// TIA Portal V17 export
// export: Created 2022-03-12T16:05:28.2107683Z, ExportSetting WithDefaults, DisplayName Totally Integrated Automation Portal, DisplayVersion V17, DisplayName TIA Portal Openness, DisplayVersion V17, DisplayName TIA Portal Version Control Interface, DisplayVersion V17, DisplayName STEP 7 Professional, DisplayVersion V17, DisplayName STEP 7 Safety, DisplayVersion V17, DisplayName WinCC Advanced / Unified PC, DisplayVersion V17
FUNCTION_BLOCK "EM01_01_EventControl"   // FB31661, LAD
TITLE = EM01_01_EventControl
{ S7_Optimized_Access := 'TRUE' }
AUTHOR : tech.team.motioncontrol@siemens.com
FAMILY : CPG
VERSION : 1.1
// Support: tech.team.motioncontrol@siemens.com
// stored: AutoNumber true, IsIECCheckEnabled false, IsRetainMemResEnabled false, MemoryReserve 100, SetENOAutomatically false, UDAEnableTagReadback false
   VAR
      instEventMgr_Alarm { ExternalAccessible := 'False'; ExternalVisible := 'False'; ExternalWritable := 'False'; S7_SetPoint := 'True'} : "CPG_EventManager";   // instance FB - Event Manager - Alarm Events
      instEventMgr_Warning { ExternalAccessible := 'False'; ExternalVisible := 'False'; ExternalWritable := 'False'; S7_SetPoint := 'True'} : "CPG_EventManager";   // instance FB - Event Manager - Warning Events
      instEventMgr_Status { ExternalAccessible := 'False'; ExternalVisible := 'False'; ExternalWritable := 'False'; S7_SetPoint := 'True'} : "CPG_EventManager";   // instance FB - Event Manager - Status Events
      instStatus_AlarmNotReset { ExternalAccessible := 'False'; ExternalVisible := 'False'; ExternalWritable := 'False'; S7_SetPoint := 'True'} : "CPG_Event";   // instance FB - PackML Event - Alarms not reset
      statEventMgr_Cmd_Reset { ExternalAccessible := 'False'; ExternalVisible := 'False'; ExternalWritable := 'False'} : Bool;   // Reset Cmd for all event managers
      statEventMgr_Cmd_Clear1stFlt { ExternalAccessible := 'False'; ExternalVisible := 'False'; ExternalWritable := 'False'} : Bool;   // Clear 1st Fault Cmd for all event managers
      statEventMgr_Clear1stFlt_OS { ExternalAccessible := 'False'; ExternalVisible := 'False'; ExternalWritable := 'False'} : Bool;   // Clear 1st Fault Cmd - One shot
   END_VAR
   VAR_TEMP   // added for the SCL form of the ladder/FBD networks
      _w1 : Bool;
      _w2 : Bool;
   END_VAR
BEGIN

REGION Network 1: ** STATE MODEL REPORTING STATUS ****
END_REGION

REGION Network 2: *** Call the PackML Module Initialize Logic ***
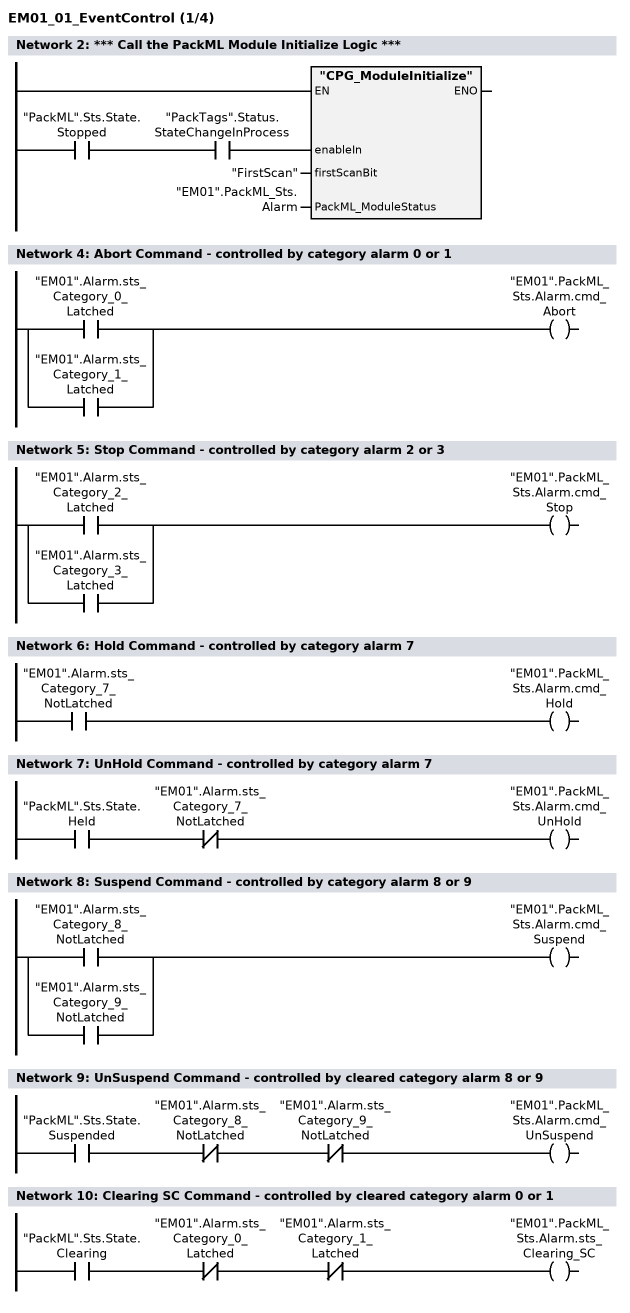
   RUNG wire#powerrail
      "CPG_ModuleInitialize"(enableIn := wire#w1, firstScanBit := "FirstScan", PackML_ModuleStatus := "EM01".PackML_Sts.Alarm)
   END_RUNG
   RUNG wire#powerrail
      Contact( "PackML".Sts.State.Stopped )
      Contact( "PackTags".Status.StateChangeInProcess )
   END_RUNG wire#w1
   // the same network as SCL:
   "CPG_ModuleInitialize"(enableIn := "PackML".Sts.State.Stopped AND "PackTags".Status.StateChangeInProcess,
                          firstScanBit := "FirstScan",
                          PackML_ModuleStatus := "EM01".PackML_Sts.Alarm);
END_REGION

REGION Network 3: Begin the LOGIC section.
END_REGION

REGION Network 4: Abort Command - controlled by category alarm 0 or 1
   RUNG wire#powerrail
      Contact( "EM01".Alarm.sts_Category_0_Latched )
      wire#w1
      Coil( "EM01".PackML_Sts.Alarm.cmd_Abort )
   END_RUNG
   RUNG wire#powerrail
      Contact( "EM01".Alarm.sts_Category_1_Latched )
   END_RUNG wire#w1
   // the same network as SCL:
   "EM01".PackML_Sts.Alarm.cmd_Abort := "EM01".Alarm.sts_Category_0_Latched OR "EM01".Alarm.sts_Category_1_Latched;
END_REGION

REGION Network 5: Stop Command - controlled by category alarm 2 or 3
   RUNG wire#powerrail
      Contact( "EM01".Alarm.sts_Category_2_Latched )
      wire#w1
      Coil( "EM01".PackML_Sts.Alarm.cmd_Stop )
   END_RUNG
   RUNG wire#powerrail
      Contact( "EM01".Alarm.sts_Category_3_Latched )
   END_RUNG wire#w1
   // the same network as SCL:
   "EM01".PackML_Sts.Alarm.cmd_Stop := "EM01".Alarm.sts_Category_2_Latched OR "EM01".Alarm.sts_Category_3_Latched;
END_REGION

REGION Network 6: Hold Command - controlled by category alarm 7
   RUNG wire#powerrail
      Contact( "EM01".Alarm.sts_Category_7_NotLatched )
      Coil( "EM01".PackML_Sts.Alarm.cmd_Hold )
   END_RUNG
   // the same network as SCL:
   "EM01".PackML_Sts.Alarm.cmd_Hold := "EM01".Alarm.sts_Category_7_NotLatched;
END_REGION

REGION Network 7: UnHold Command - controlled by category alarm 7
   RUNG wire#powerrail
      Contact( "PackML".Sts.State.Held )
      I_Contact( "EM01".Alarm.sts_Category_7_NotLatched )
      Coil( "EM01".PackML_Sts.Alarm.cmd_UnHold )
   END_RUNG
   // the same network as SCL:
   "EM01".PackML_Sts.Alarm.cmd_UnHold := "PackML".Sts.State.Held AND NOT "EM01".Alarm.sts_Category_7_NotLatched;
END_REGION

REGION Network 8: Suspend Command - controlled by category alarm 8 or 9
   RUNG wire#powerrail
      Contact( "EM01".Alarm.sts_Category_8_NotLatched )
      wire#w1
      Coil( "EM01".PackML_Sts.Alarm.cmd_Suspend )
   END_RUNG
   RUNG wire#powerrail
      Contact( "EM01".Alarm.sts_Category_9_NotLatched )
   END_RUNG wire#w1
   // the same network as SCL:
   "EM01".PackML_Sts.Alarm.cmd_Suspend := "EM01".Alarm.sts_Category_8_NotLatched OR "EM01".Alarm.sts_Category_9_NotLatched;
END_REGION

REGION Network 9: UnSuspend Command - controlled by cleared category alarm 8 or 9
   RUNG wire#powerrail
      Contact( "PackML".Sts.State.Suspended )
      I_Contact( "EM01".Alarm.sts_Category_8_NotLatched )
      I_Contact( "EM01".Alarm.sts_Category_9_NotLatched )
      Coil( "EM01".PackML_Sts.Alarm.cmd_UnSuspend )
   END_RUNG
   // the same network as SCL:
   "EM01".PackML_Sts.Alarm.cmd_UnSuspend := "PackML".Sts.State.Suspended AND NOT "EM01".Alarm.sts_Category_8_NotLatched AND NOT "EM01".Alarm.sts_Category_9_NotLatched;
END_REGION

REGION Network 10: Clearing SC Command - controlled by cleared category alarm 0 or 1
   RUNG wire#powerrail
      Contact( "PackML".Sts.State.Clearing )
      I_Contact( "EM01".Alarm.sts_Category_0_Latched )
      I_Contact( "EM01".Alarm.sts_Category_1_Latched )
      Coil( "EM01".PackML_Sts.Alarm.sts_Clearing_SC )
   END_RUNG
   // the same network as SCL:
   "EM01".PackML_Sts.Alarm.sts_Clearing_SC := "PackML".Sts.State.Clearing AND NOT "EM01".Alarm.sts_Category_0_Latched AND NOT "EM01".Alarm.sts_Category_1_Latched;
END_REGION

REGION Network 11: Resetting SC Command - controlled by cleared category alarm 0-3
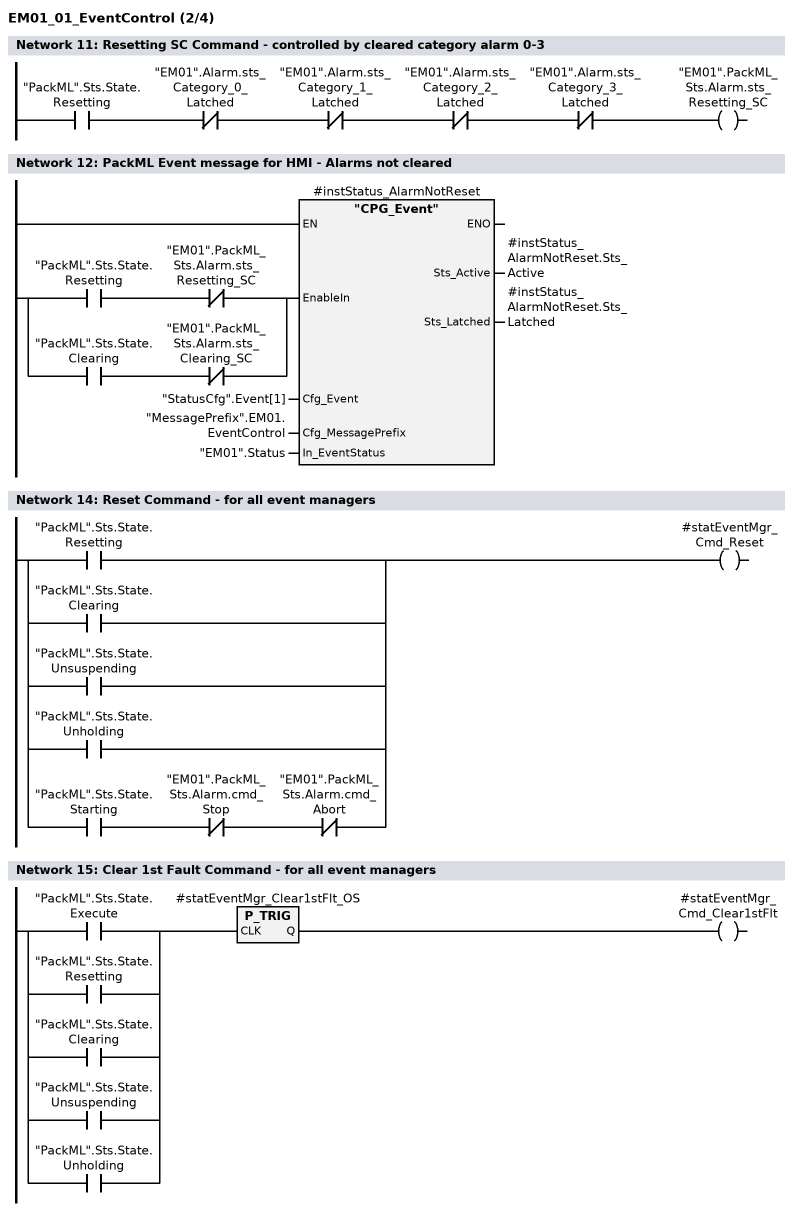
   RUNG wire#powerrail
      Contact( "PackML".Sts.State.Resetting )
      I_Contact( "EM01".Alarm.sts_Category_0_Latched )
      I_Contact( "EM01".Alarm.sts_Category_1_Latched )
      I_Contact( "EM01".Alarm.sts_Category_2_Latched )
      I_Contact( "EM01".Alarm.sts_Category_3_Latched )
      Coil( "EM01".PackML_Sts.Alarm.sts_Resetting_SC )
   END_RUNG
   // the same network as SCL:
   "EM01".PackML_Sts.Alarm.sts_Resetting_SC := "PackML".Sts.State.Resetting AND NOT "EM01".Alarm.sts_Category_0_Latched AND NOT "EM01".Alarm.sts_Category_1_Latched AND NOT "EM01".Alarm.sts_Category_2_Latched AND NOT "EM01".Alarm.sts_Category_3_Latched;
END_REGION

REGION Network 12: PackML Event message for HMI - Alarms not cleared
   RUNG wire#powerrail
      #instStatus_AlarmNotReset(EnableIn := wire#w1, Cfg_Event := "StatusCfg".Event[1], Cfg_MessagePrefix := "MessagePrefix".EM01.EventControl, In_EventStatus := "EM01".Status, Sts_Active => #instStatus_AlarmNotReset.Sts_Active, Sts_Latched => #instStatus_AlarmNotReset.Sts_Latched)
   END_RUNG
   RUNG wire#powerrail
      Contact( "PackML".Sts.State.Resetting )
      I_Contact( "EM01".PackML_Sts.Alarm.sts_Resetting_SC )
   END_RUNG wire#w1
   RUNG wire#powerrail
      Contact( "PackML".Sts.State.Clearing )
      I_Contact( "EM01".PackML_Sts.Alarm.sts_Clearing_SC )
   END_RUNG wire#w1
   // the same network as SCL:
   #instStatus_AlarmNotReset(EnableIn := ("PackML".Sts.State.Resetting AND NOT "EM01".PackML_Sts.Alarm.sts_Resetting_SC) OR ("PackML".Sts.State.Clearing AND NOT "EM01".PackML_Sts.Alarm.sts_Clearing_SC),   // "CPG_Event"
                           Cfg_Event := "StatusCfg".Event[1],
                           Cfg_MessagePrefix := "MessagePrefix".EM01.EventControl,
                           In_EventStatus := "EM01".Status,
                           Sts_Active => #instStatus_AlarmNotReset.Sts_Active,
                           Sts_Latched => #instStatus_AlarmNotReset.Sts_Latched);
END_REGION

REGION Network 13: *** EVENT CONTROL MANAGERS ***
END_REGION

REGION Network 14: Reset Command - for all event managers
   RUNG wire#powerrail
      Contact( "PackML".Sts.State.Resetting )
      wire#w1
      Coil( #statEventMgr_Cmd_Reset )
   END_RUNG
   RUNG wire#powerrail
      Contact( "PackML".Sts.State.Clearing )
   END_RUNG wire#w1
   RUNG wire#powerrail
      Contact( "PackML".Sts.State.Unsuspending )
   END_RUNG wire#w1
   RUNG wire#powerrail
      Contact( "PackML".Sts.State.Unholding )
   END_RUNG wire#w1
   RUNG wire#powerrail
      Contact( "PackML".Sts.State.Starting )
      I_Contact( "EM01".PackML_Sts.Alarm.cmd_Stop )
      I_Contact( "EM01".PackML_Sts.Alarm.cmd_Abort )
   END_RUNG wire#w1
   // the same network as SCL:
   #statEventMgr_Cmd_Reset := "PackML".Sts.State.Resetting OR "PackML".Sts.State.Clearing OR "PackML".Sts.State.Unsuspending OR "PackML".Sts.State.Unholding OR ("PackML".Sts.State.Starting AND NOT "EM01".PackML_Sts.Alarm.cmd_Stop AND NOT "EM01".PackML_Sts.Alarm.cmd_Abort);
END_REGION

REGION Network 15: Clear 1st Fault Command - for all event managers
   RUNG wire#powerrail
      Contact( "PackML".Sts.State.Execute )
      wire#w1
      P_Trig( #statEventMgr_Clear1stFlt_OS )
      Coil( #statEventMgr_Cmd_Clear1stFlt )
   END_RUNG
   RUNG wire#powerrail
      Contact( "PackML".Sts.State.Resetting )
   END_RUNG wire#w1
   RUNG wire#powerrail
      Contact( "PackML".Sts.State.Clearing )
   END_RUNG wire#w1
   RUNG wire#powerrail
      Contact( "PackML".Sts.State.Unsuspending )
   END_RUNG wire#w1
   RUNG wire#powerrail
      Contact( "PackML".Sts.State.Unholding )
   END_RUNG wire#w1
   // the same network as SCL:
   #_w1 := "PackML".Sts.State.Execute OR "PackML".Sts.State.Resetting OR "PackML".Sts.State.Clearing OR "PackML".Sts.State.Unsuspending OR "PackML".Sts.State.Unholding;
   #_w2 := #_w1 AND NOT #statEventMgr_Clear1stFlt_OS;   // rising edge
   #statEventMgr_Clear1stFlt_OS := #_w1;
   #statEventMgr_Cmd_Clear1stFlt := #_w2;
END_REGION

REGION Network 16: Call the Event Manager logic for EM alarms
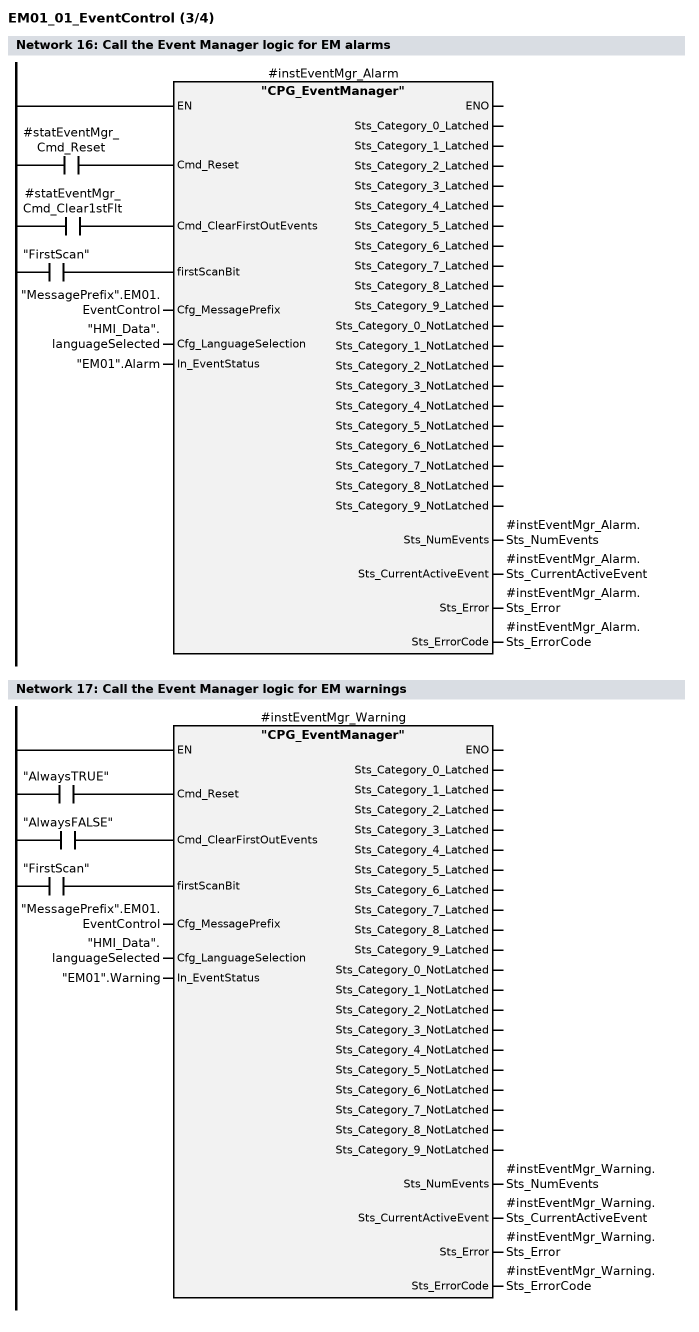
   RUNG wire#powerrail
      #instEventMgr_Alarm(Cmd_Reset := wire#w1, Cmd_ClearFirstOutEvents := wire#w2, firstScanBit := wire#w3, Cfg_MessagePrefix := "MessagePrefix".EM01.EventControl, Cfg_LanguageSelection := "HMI_Data".languageSelected, In_EventStatus := "EM01".Alarm, Sts_Category_0_Latched =>, Sts_Category_1_Latched =>, Sts_Category_2_Latched =>, Sts_Category_3_Latched =>, Sts_Category_4_Latched =>, Sts_Category_5_Latched =>, Sts_Category_6_Latched =>, Sts_Category_7_Latched =>, Sts_Category_8_Latched =>, Sts_Category_9_Latched =>, Sts_Category_0_NotLatched =>, Sts_Category_1_NotLatched =>, Sts_Category_2_NotLatched =>, Sts_Category_3_NotLatched =>, Sts_Category_4_NotLatched =>, Sts_Category_5_NotLatched =>, Sts_Category_6_NotLatched =>, Sts_Category_7_NotLatched =>, Sts_Category_8_NotLatched =>, Sts_Category_9_NotLatched =>, Sts_NumEvents => #instEventMgr_Alarm.Sts_NumEvents, Sts_CurrentActiveEvent => #instEventMgr_Alarm.Sts_CurrentActiveEvent, Sts_Error => #instEventMgr_Alarm.Sts_Error, Sts_ErrorCode => #instEventMgr_Alarm.Sts_ErrorCode)
   END_RUNG
   RUNG wire#powerrail
      Contact( #statEventMgr_Cmd_Reset )
   END_RUNG wire#w1
   RUNG wire#powerrail
      Contact( #statEventMgr_Cmd_Clear1stFlt )
   END_RUNG wire#w2
   RUNG wire#powerrail
      Contact( "FirstScan" )
   END_RUNG wire#w3
   // the same network as SCL:
   #instEventMgr_Alarm(Cmd_Reset := #statEventMgr_Cmd_Reset,   // "CPG_EventManager"
                       Cmd_ClearFirstOutEvents := #statEventMgr_Cmd_Clear1stFlt,
                       firstScanBit := "FirstScan",
                       Cfg_MessagePrefix := "MessagePrefix".EM01.EventControl,
                       Cfg_LanguageSelection := "HMI_Data".languageSelected,
                       In_EventStatus := "EM01".Alarm,
                       Sts_NumEvents => #instEventMgr_Alarm.Sts_NumEvents,
                       Sts_CurrentActiveEvent => #instEventMgr_Alarm.Sts_CurrentActiveEvent,
                       Sts_Error => #instEventMgr_Alarm.Sts_Error,
                       Sts_ErrorCode => #instEventMgr_Alarm.Sts_ErrorCode);
END_REGION

REGION Network 17: Call the Event Manager logic for EM warnings
   RUNG wire#powerrail
      #instEventMgr_Warning(Cmd_Reset := wire#w1, Cmd_ClearFirstOutEvents := wire#w2, firstScanBit := wire#w3, Cfg_MessagePrefix := "MessagePrefix".EM01.EventControl, Cfg_LanguageSelection := "HMI_Data".languageSelected, In_EventStatus := "EM01".Warning, Sts_Category_0_Latched =>, Sts_Category_1_Latched =>, Sts_Category_2_Latched =>, Sts_Category_3_Latched =>, Sts_Category_4_Latched =>, Sts_Category_5_Latched =>, Sts_Category_6_Latched =>, Sts_Category_7_Latched =>, Sts_Category_8_Latched =>, Sts_Category_9_Latched =>, Sts_Category_0_NotLatched =>, Sts_Category_1_NotLatched =>, Sts_Category_2_NotLatched =>, Sts_Category_3_NotLatched =>, Sts_Category_4_NotLatched =>, Sts_Category_5_NotLatched =>, Sts_Category_6_NotLatched =>, Sts_Category_7_NotLatched =>, Sts_Category_8_NotLatched =>, Sts_Category_9_NotLatched =>, Sts_NumEvents => #instEventMgr_Warning.Sts_NumEvents, Sts_CurrentActiveEvent => #instEventMgr_Warning.Sts_CurrentActiveEvent, Sts_Error => #instEventMgr_Warning.Sts_Error, Sts_ErrorCode => #instEventMgr_Warning.Sts_ErrorCode)
   END_RUNG
   RUNG wire#powerrail
      Contact( "AlwaysTRUE" )
   END_RUNG wire#w1
   RUNG wire#powerrail
      Contact( "AlwaysFALSE" )
   END_RUNG wire#w2
   RUNG wire#powerrail
      Contact( "FirstScan" )
   END_RUNG wire#w3
   // the same network as SCL:
   #instEventMgr_Warning(Cmd_Reset := "AlwaysTRUE",   // "CPG_EventManager"
                         Cmd_ClearFirstOutEvents := "AlwaysFALSE",
                         firstScanBit := "FirstScan",
                         Cfg_MessagePrefix := "MessagePrefix".EM01.EventControl,
                         Cfg_LanguageSelection := "HMI_Data".languageSelected,
                         In_EventStatus := "EM01".Warning,
                         Sts_NumEvents => #instEventMgr_Warning.Sts_NumEvents,
                         Sts_CurrentActiveEvent => #instEventMgr_Warning.Sts_CurrentActiveEvent,
                         Sts_Error => #instEventMgr_Warning.Sts_Error,
                         Sts_ErrorCode => #instEventMgr_Warning.Sts_ErrorCode);
END_REGION

REGION Network 18: Call the Event Manager logic for EM status
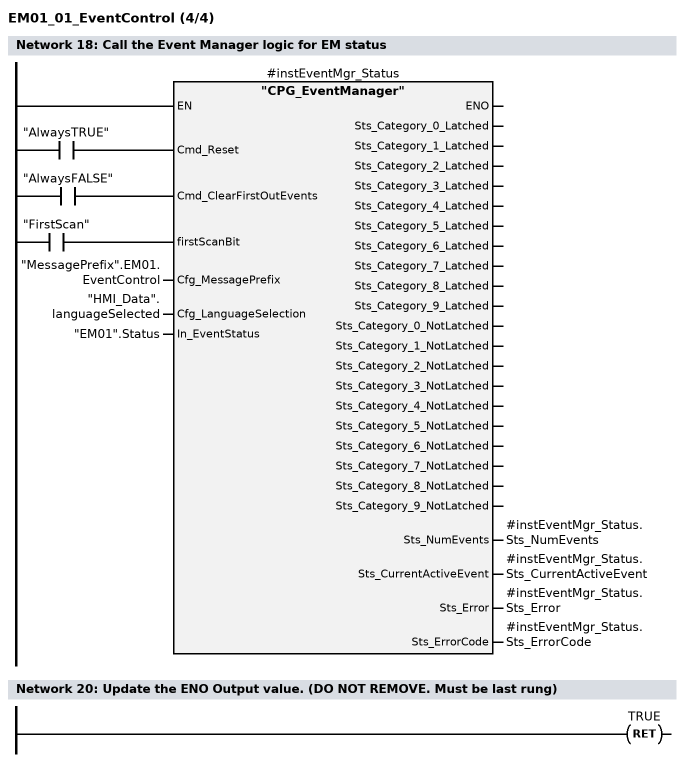
   RUNG wire#powerrail
      #instEventMgr_Status(Cmd_Reset := wire#w1, Cmd_ClearFirstOutEvents := wire#w2, firstScanBit := wire#w3, Cfg_MessagePrefix := "MessagePrefix".EM01.EventControl, Cfg_LanguageSelection := "HMI_Data".languageSelected, In_EventStatus := "EM01".Status, Sts_Category_0_Latched =>, Sts_Category_1_Latched =>, Sts_Category_2_Latched =>, Sts_Category_3_Latched =>, Sts_Category_4_Latched =>, Sts_Category_5_Latched =>, Sts_Category_6_Latched =>, Sts_Category_7_Latched =>, Sts_Category_8_Latched =>, Sts_Category_9_Latched =>, Sts_Category_0_NotLatched =>, Sts_Category_1_NotLatched =>, Sts_Category_2_NotLatched =>, Sts_Category_3_NotLatched =>, Sts_Category_4_NotLatched =>, Sts_Category_5_NotLatched =>, Sts_Category_6_NotLatched =>, Sts_Category_7_NotLatched =>, Sts_Category_8_NotLatched =>, Sts_Category_9_NotLatched =>, Sts_NumEvents => #instEventMgr_Status.Sts_NumEvents, Sts_CurrentActiveEvent => #instEventMgr_Status.Sts_CurrentActiveEvent, Sts_Error => #instEventMgr_Status.Sts_Error, Sts_ErrorCode => #instEventMgr_Status.Sts_ErrorCode)
   END_RUNG
   RUNG wire#powerrail
      Contact( "AlwaysTRUE" )
   END_RUNG wire#w1
   RUNG wire#powerrail
      Contact( "AlwaysFALSE" )
   END_RUNG wire#w2
   RUNG wire#powerrail
      Contact( "FirstScan" )
   END_RUNG wire#w3
   // the same network as SCL:
   #instEventMgr_Status(Cmd_Reset := "AlwaysTRUE",   // "CPG_EventManager"
                        Cmd_ClearFirstOutEvents := "AlwaysFALSE",
                        firstScanBit := "FirstScan",
                        Cfg_MessagePrefix := "MessagePrefix".EM01.EventControl,
                        Cfg_LanguageSelection := "HMI_Data".languageSelected,
                        In_EventStatus := "EM01".Status,
                        Sts_NumEvents => #instEventMgr_Status.Sts_NumEvents,
                        Sts_CurrentActiveEvent => #instEventMgr_Status.Sts_CurrentActiveEvent,
                        Sts_Error => #instEventMgr_Status.Sts_Error,
                        Sts_ErrorCode => #instEventMgr_Status.Sts_ErrorCode);
END_REGION

REGION Network 20: Update the ENO Output value. (DO NOT REMOVE. Must be last rung)
   RUNG wire#powerrail
      ReturnCoil( TRUE )
   END_RUNG
   // the same network as SCL:
   ENO := TRUE;
   RETURN;
END_REGION
END_FUNCTION_BLOCK
